FUNCTION_BLOCK PLOT_CALLBACK
  {SET_ATTRIBUTE(OpcUa, SERVICE)}
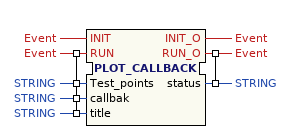
  EVENT_INPUT
    INIT;
    RUN WITH Test_points, callbak, title; {SET_ATTRIBUTE(OpcUa, Method)}
  END_EVENT
  EVENT_OUTPUT
    INIT_O;
    RUN_O WITH status;
  END_EVENT
  VAR_INPUT
    Test_points : STRING; {SET_ATTRIBUTE(OpcUa, Variable.RUN)}
    callbak : STRING; {SET_ATTRIBUTE(OpcUa, Variable.RUN)}
    title : STRING; {SET_ATTRIBUTE(OpcUa, Variable.RUN)}
  END_VAR
  VAR_OUTPUT
    status : STRING; {SET_ATTRIBUTE(OpcUa, Variable.RUN)}
  END_VAR
END_FUNCTION_BLOCK
